{attribute 'GeneratedUsingTerminal: EL3011-0000-0016'}
{attribute addProperty BoxType "EL3011-0000-0016"}
{attribute addProperty Description "EL3011 4Ch. Ana. Input 0-20mA DIFF"}
{attribute addProperty Physics "KK"}
{attribute addProperty Id "AI_StandardAT %I*AI_Standard_Channel_4A3944819WcStateAT %I*WcState_9091E0EB2InfoDataAT %I*InfoData_32EB74EA10"}
{attribute addProperty CRC "3794663976"}
{attribute addProperty Size "21"}
TYPE EL3011_E22DFA28 EXTENDS EtcSlaveTerminalBase_947E5A46 :
STRUCT
	{attribute addProperty Name "AI_Standard"}
	AI_Standard : AI_Standard_Channel_4A394481;
	{attribute addProperty Name "WcState"}
	WcState : WcState_9091E0EB;
	{attribute addProperty Name "InfoData"}
	InfoData : InfoData_32EB74EA;
END_STRUCT
END_TYPE

(* stored: Version 1.2.0.0, ProductVersion 3.1.4024.11
   DUT EL3011_E22DFA28: Id {676d68eb-0e61-4ea7-864a-3bd621d46711} *)
